// Block: DEBUG

DATA_BLOCK DEBUG
VERSION : 0.1
   NON_RETAIN
   VAR
      Force_Sinamics_Infeed_ON : Bool;
      Alr : Array[1..10] of Bool;
      Core_iSlaveSynchPos : LReal;
      "Core.iMasterSyncPos" : LReal;
      "Core.iWorkPosition" : LReal;
      "Core.SlavePosition" : LReal;
   END_VAR

BEGIN
   // No initialization required
END_DATA_BLOCK
